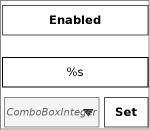
VISUALIZATION vHP3_AxisBrakeControl  // 150x130
VAR_IN_OUT
	fbData	: fbHP_Axis;
END_VAR
    Rectangle (104,97 44x30), "Set", colour toggle: fbData.bSetNewBrakeCtrl, input disabled if: NOT fbData.ManualMode
        toggle fbData.bSetNewBrakeCtrl p2164770859=TRUE
    Rectangle (2,5 146x30), "Enabled", colour toggle: fbData.Enabled, input disabled if: NOT fbData.ManualMode
        toggle fbData.bTooglePowerState
    Rectangle (2,57 146x30), "%s", text variable: TO_STRING(fbData.nAct_BrakeMode)
    ComboBoxInteger (4,97 95x30), variable: fbData.nNew_BrakeMode, input disabled if: NOT fbData.ManualMode
END_VISUALIZATION

(* stored: Version 1.1.0.1, ProductVersion 3.1.4024.12
   Visu vHP3_AxisBrakeControl: Id {0ffd8913-1a96-456f-a29c-931ee95cd276} *)
